FUNCTION_BLOCK FB_SPR
VAR_INPUT
END_VAR
VAR_OUTPUT
END_VAR
VAR
	Pufferspeicher_Kaltwasser_195						: FB_PSp;
	Pufferspeicher_Warmwasser_295						: FB_PSp;
	Pufferspeicher_Heisswasser_395						: FB_PSp;
	System_Betonspeicher_Kaltwasser_795					: FB_System_BSp_795;
	System_Betonspeicher_Warmwasser_797					: FB_System_BSp_797;
END_VAR

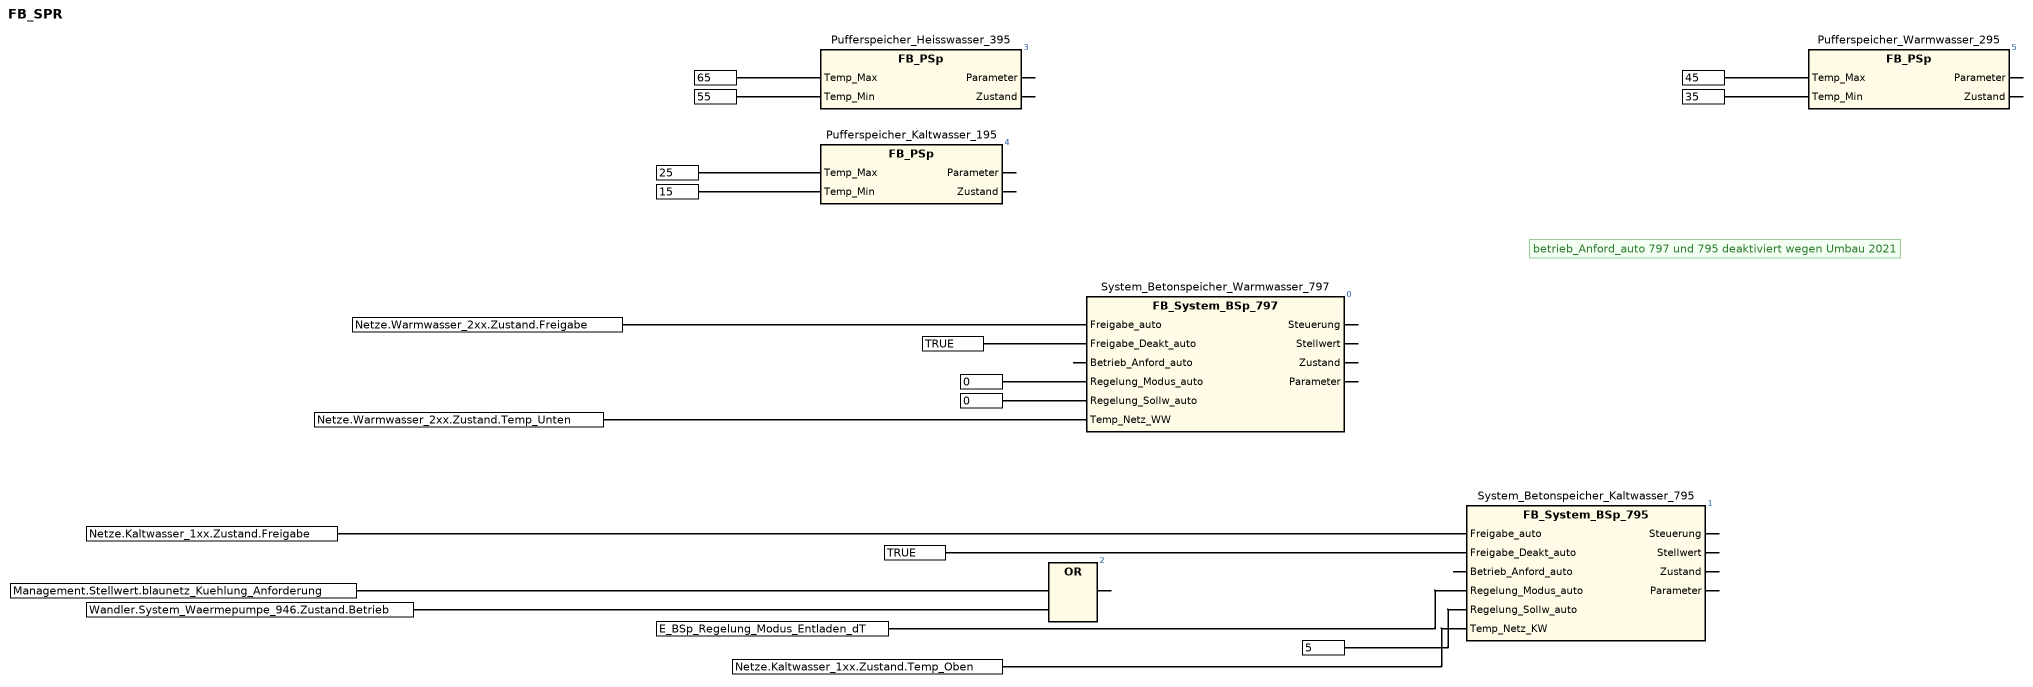
// betrieb_Anford_auto 797 und 795 deaktiviert wegen Umbau 2021
System_Betonspeicher_Warmwasser_797(
    Freigabe_auto := Netze.Warmwasser_2xx.Zustand.Freigabe,
    Freigabe_Deakt_auto := TRUE,
    Regelung_Modus_auto := 0,
    Regelung_Sollw_auto := 0,
    Temp_Netz_WW := Netze.Warmwasser_2xx.Zustand.Temp_Unten); // FB_System_BSp_797
System_Betonspeicher_Kaltwasser_795(
    Freigabe_auto := Netze.Kaltwasser_1xx.Zustand.Freigabe,
    Freigabe_Deakt_auto := TRUE,
    Regelung_Modus_auto := E_BSp_Regelung_Modus_Entladen_dT,
    Regelung_Sollw_auto := 5,
    Temp_Netz_KW := Netze.Kaltwasser_1xx.Zustand.Temp_Oben); // FB_System_BSp_795
(* Management.Stellwert.blaunetz_Kuehlung_Anforderung OR Wandler.System_Waermepumpe_946.Zustand.Betrieb; result not used *)
Pufferspeicher_Heisswasser_395(Temp_Max := 65, Temp_Min := 55); // FB_PSp
Pufferspeicher_Kaltwasser_195(Temp_Max := 25, Temp_Min := 15); // FB_PSp
Pufferspeicher_Warmwasser_295(Temp_Max := 45, Temp_Min := 35); // FB_PSp

END_FUNCTION_BLOCK

(* stored: Version 1.1.0.1, ProductVersion 3.1.4024.9
   POU FB_SPR: Id {533d91c1-442a-403a-a6ee-f4dbb832db78}, SpecialFunc None *)
